% RSLogix 500 project PLC1_Lesson_6_Lab_2.RSS, saved by version 12.00.00.00 %
PROJECT "UNTITLED"    % processor: Bul.1763 MicroLogix 1100 Series B %

PROGRAM FILES
  LAD 2   3 rungs

DATA FILES
  O0 OUTPUT  5 elements
  I1 INPUT  6 elements
  S2 STATUS  66 elements
  B3 BINARY  1 elements
  T4 TIMER  2 elements
  C5 COUNTER  1 elements
  R6 CONTROL  1 elements
  N7 INTEGER  1 elements
  F8 FLOAT  1 elements

LADDER 2
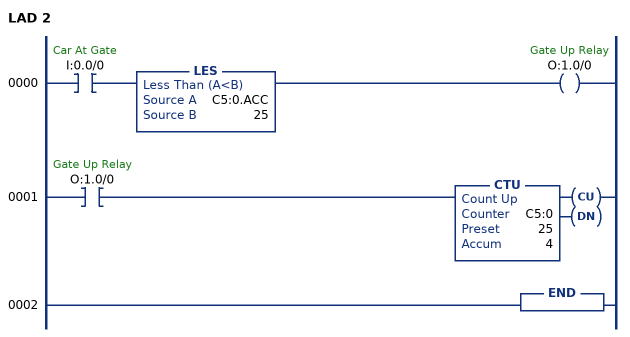
% Rung: 0 %
SOR XIC I:0.0/0 LES C5:0.ACC 25 OTE O:1.0/0 EOR
%   I:0.0/0  "Car At Gate" %
%   O:1.0/0  "Gate Up Relay" %
% Rung: 1 %
SOR XIC O:1.0/0 CTU C5:0 25 4 EOR
%   O:1.0/0  "Gate Up Relay" %
% Rung: 2 %
SOR END EOR

DATA TABLE (non-zero values as saved)
DATA T4
% .PRE .ACC %
% T4:0 % 5 0
% T4:1 % 5 5
DATA C5
% .PRE .ACC %
% C5:0 % 25 4
